TYPE HLSInputs :
STRUCT
	iIn : INT;
END_STRUCT
END_TYPE

(* stored: Version 1.1.0.1, ProductVersion 3.1.4024.12
   DUT HLSInputs: Id {b2d86cbb-e3cc-4dc9-98e0-50e036370629} *)
